INTERFACE I_PidController

PROPERTY Deviation : BOOL
GET
END_GET
END_PROPERTY

PROPERTY Enable : BOOL
GET
END_GET
SET
END_SET
END_PROPERTY

PROPERTY Error : BOOL
GET
END_GET
END_PROPERTY

METHOD Exectute
VAR_INPUT
	fSetpointValue	: LREAL;
	fProcessValue	: LREAL;
END_VAR
END_METHOD

PROPERTY Overrange : BOOL
GET
END_GET
END_PROPERTY

PROPERTY PidParameters : REFERENCE TO ST_PidControllerParameters
GET
END_GET
SET
END_SET
END_PROPERTY

METHOD Reset
VAR_INPUT
END_VAR
END_METHOD

PROPERTY Underrange : BOOL
GET
END_GET
END_PROPERTY

END_INTERFACE

(* stored: Version 1.1.0.1, ProductVersion 3.1.4024.13
   Itf I_PidController: Id {0e4ab069-6ce9-0f17-3ba3-5874e6414979}
   Property Deviation: Id {9b2d2a3b-0831-0d6c-3032-73a0b71521f4}
   Get Get: Id {426db43d-8009-0eb8-2146-a2894a1e101d}
   Property Enable: Id {fe824e5a-5005-02cb-0e17-3a605287a4b0}
   Get Get: Id {4df5c014-b80c-05c8-1bb0-5bf1462e0b4f}
   Set Set: Id {23ecba45-bed6-03ac-1902-7ba3f7e2879d}
   Property Error: Id {da7ddbe6-439b-09c9-1d82-08d70eecfbb1}
   Get Get: Id {8f64b220-9568-0330-27fd-8aaa8c19024e}
   Method Exectute: Id {58665bec-c176-06d3-1b12-64b4a4edbd1d}
   Property Overrange: Id {5f75845e-edf4-018d-2422-2b44b0981b8c}
   Get Get: Id {1fe85ad3-cd28-0dd8-1e8d-2115720204cb}
   Property PidParameters: Id {91359069-543e-027d-3ede-547fa4f2b782}
   Get Get: Id {fcc49ca6-246b-0a03-1291-ad3dbee5fb0e}
   Set Set: Id {c3364861-a884-0071-31da-ee3db34c7e80}
   Method Reset: Id {fa0bc785-fa5f-0968-1cc4-eaa081f5553f}
   Property Underrange: Id {43231de5-311d-0ec8-0e82-31565b597b95}
   Get Get: Id {9d993d70-9824-0a11-2ed7-18e5b0eac37b} *)
